GLOBALCONSTANTS DefaultPool_Scroll (* Scroll list configuration constants (geometry + controls) *)
  PACKAGE Uebungen::const::UT::Scroll;
  VAR_GLOBAL CONSTANT
    Container_Scroll : isobus::utils::scroll::ScrollFull_S := (stGeometry := (u16ListParentId := 3006, u16ListContentId := 3031, i32RowHeight := 42, u16BarParentId := 3000, u16BarContentId := 3010, i32BarBaseOffset := -252, i32BarTravel := 252, i32PosMax := 13, i32Step := 6), stControls := (u16BtnTopId := 65535, u16BtnPageUpId := 27026, u16BtnUpId := 27027, u16BtnDownId := 27028, u16BtnPageDownId := 27029, u16BtnBottomId := 65535, u16GotoInputId := 65535));
  END_VAR
END_GLOBALCONSTANTS
